(* IEC 61131-3 sources: RL_MAR/experiments/comparison/llm4plc/results/gpt-4o-mini_20260506_100619/20260506_103313, 3 files *)

(* ---- generated_code_iteration_0.st ---- *)
ructured-text
START_ST
FUNCTION_BLOCK FB_Fibonacci_Calculator
VAR_INPUT
    N : DINT := 5; // Input value for Fibonacci calculation
END_VAR
VAR_OUTPUT
    O : DINT := 1; // Output value for Fibonacci result
END_VAR
VAR
    F1 : DINT := 1; // First Fibonacci number
    F2 : DINT := 1; // Second Fibonacci number
    CNT : DINT := 2; // Counter for Fibonacci terms
    state : INT; // The state variable
END_VAR

// State Initialization
state := 0;

// State Machine Logic
WHILE TRUE DO
    CASE state OF
        0: // STATE 0: INITIALIZE
            CNT := 2;
            O := 1;
            IF N <= 2 THEN
                state := 2; // Transition to STATE 2
            ELSE
                state := 1; // Transition to STATE 1
            END_IF;

        1: // STATE 1: CALCULATE_FIBONACCI
            WHILE CNT < N DO
                VAR
                    F_next : DINT; // Next Fibonacci number
                END_VAR
                F_next := F1 + F2;
                IF F_next > 32767 THEN
                    O := 32767; // Saturation
                ELSE
                    O := F_next;
                END_IF;
                F1 := F2;
                F2 := O;
                CNT := CNT + 1;
            END_WHILE;
            state := 2; // Transition to STATE 2

        2: // STATE 2: RETURN_RESULT
            O := F2; // Set O to the final Fibonacci number
            state := 0; // Reset state for next execution
    END_CASE;
END_WHILE;

END_FUNCTION_BLOCK
END_ST

(* ---- generated_code_iteration_1.st ---- *)
START_REASON
The errors in the original Structured Text (ST) code occurred because the variable `state` was declared in the main variable section without being properly categorized. In Structured Text, all variables must be declared in the appropriate sections: VAR, VAR_INPUT, VAR_OUTPUT, or VAR_IN_OUT. The feedback specifically indicated that `state` should be declared using one of these sections, which I will correct in the improved code.
END_REASON

START_ST
FUNCTION_BLOCK FB_Fibonacci_Calculator
VAR_INPUT
    N : DINT := 5; // Input value for Fibonacci calculation
END_VAR
VAR_OUTPUT
    O : DINT := 1; // Output value for Fibonacci result
END_VAR
VAR
    F1 : DINT := 1; // First Fibonacci number
    F2 : DINT := 1; // Second Fibonacci number
    CNT : DINT := 2; // Counter for Fibonacci terms
    state : INT := 0; // The state variable initialized to 0
END_VAR

// State Machine Logic
WHILE TRUE DO
    CASE state OF
        0: // STATE 0: INITIALIZE
            CNT := 2;
            O := 1;
            IF N <= 2 THEN
                state := 2; // Transition to STATE 2
            ELSE
                state := 1; // Transition to STATE 1
            END_IF;

        1: // STATE 1: CALCULATE_FIBONACCI
            WHILE CNT < N DO
                VAR
                    F_next : DINT; // Next Fibonacci number
                END_VAR
                F_next := F1 + F2;
                IF F_next > 32767 THEN
                    O := 32767; // Saturation
                ELSE
                    O := F_next;
                END_IF;
                F1 := F2;
                F2 := O;
                CNT := CNT + 1;
            END_WHILE;
            state := 2; // Transition to STATE 2

        2: // STATE 2: RETURN_RESULT
            O := F2; // Set O to the final Fibonacci number
            state := 0; // Reset state for next execution
    END_CASE;
END_WHILE;

END_FUNCTION_BLOCK
END_ST

(* ---- generated_code_iteration_2.st ---- *)
START_REASON
The errors in the original Structured Text (ST) code occurred due to the improper placement of the variable declaration for `F_next` inside the `WHILE` loop. In Structured Text, variable declarations should be placed in the appropriate variable sections and not within control structures like loops or conditionals. This caused the code to fail during compilation. I will correct this by moving the declaration of `F_next` to the main variable section and ensuring that the overall structure adheres to the rules of Structured Text.
END_REASON

START_ST
FUNCTION_BLOCK FB_Fibonacci_Calculator
VAR_INPUT
    N : DINT := 5; // Input value for Fibonacci calculation
END_VAR
VAR_OUTPUT
    O : DINT := 1; // Output value for Fibonacci result
END_VAR
VAR
    F1 : DINT := 1; // First Fibonacci number
    F2 : DINT := 1; // Second Fibonacci number
    CNT : DINT := 2; // Counter for Fibonacci terms
    state : INT := 0; // The state variable initialized to 0
    F_next : DINT; // Next Fibonacci number
END_VAR

// State Machine Logic
WHILE TRUE DO
    CASE state OF
        0: // STATE 0: INITIALIZE
            CNT := 2;
            O := 1;
            IF N <= 2 THEN
                state := 2; // Transition to STATE 2
            ELSE
                state := 1; // Transition to STATE 1
            END_IF;

        1: // STATE 1: CALCULATE_FIBONACCI
            WHILE CNT < N DO
                F_next := F1 + F2;
                IF F_next > 32767 THEN
                    O := 32767; // Saturation
                ELSE
                    O := F_next;
                END_IF;
                F1 := F2;
                F2 := O;
                CNT := CNT + 1;
            END_WHILE;
            state := 2; // Transition to STATE 2

        2: // STATE 2: RETURN_RESULT
            O := F2; // Set O to the final Fibonacci number
            state := 0; // Reset state for next execution
    END_CASE;
END_WHILE;

END_FUNCTION_BLOCK
END_ST
